// TIA Portal V15.1 export
// export: Created 2024-05-17T05:38:40.3336056Z, ExportSetting WithDefaults, DisplayName Totally Integrated Automation Portal, DisplayVersion V15.1 Update 5, DisplayName TIA Portal Openness, DisplayVersion V15.1 Update 5, DisplayName SINAMICS Startdrive Advanced, DisplayVersion V15.1, DisplayName G130, G150, S120, S150, SINAMICS MV, S210, DisplayVersion V15.1, DisplayName G110M, G120, G120C, G120D, G120P, DisplayVersion V15.1, DisplayName STEP 7 Professional, DisplayVersion V15.1 Update 5, DisplayName STEP 7 Safety, DisplayVersion V15.1, DisplayName WinCC Professional, DisplayVersion V15.1 Update 5, DisplayName SIMATIC Visualization Architect, DisplayVersion V15.1
FUNCTION "LGBHWPanelLedIndication" : Void   // FC6610, FBD
TITLE = LGBHWPanelLedIndication
{ S7_Optimized_Access := 'TRUE' }
VERSION : 0.1
// stored: AutoNumber false, IsIECCheckEnabled false, SetENOAutomatically False, UDAEnableTagReadback false
   VAR_INPUT
      I_NumberHMI : Int;   // Number of this HMI in the Modeselector
      I_ActiveHMI : Int;   // Active HMI in the Modeselector
      I_EStopAS_OK : Bool;   // Emergency Stop On AS Panel
      I_EStopZone_OK : Bool;   // Emergency Stop In The Safety Zone
      I_AlarmA : Bool;   // AlarmA
      I_AlarmB : Bool;   // AlarmB
      I_AlarmC : Bool;   // AlarmC
      I_Modes : "Modes";   // Modes
   END_VAR
   VAR_OUTPUT
      O_LED_Auto : Bool;   // Indication Automatic
      O_LED_Man : Bool;   // Indication Manual
      O_LED_Fault : Bool;   // Indication Fault
      O_LED_EStop : Bool;   // Indication Emergency Stop
   END_VAR
BEGIN

REGION Network 1: Indication Automatic
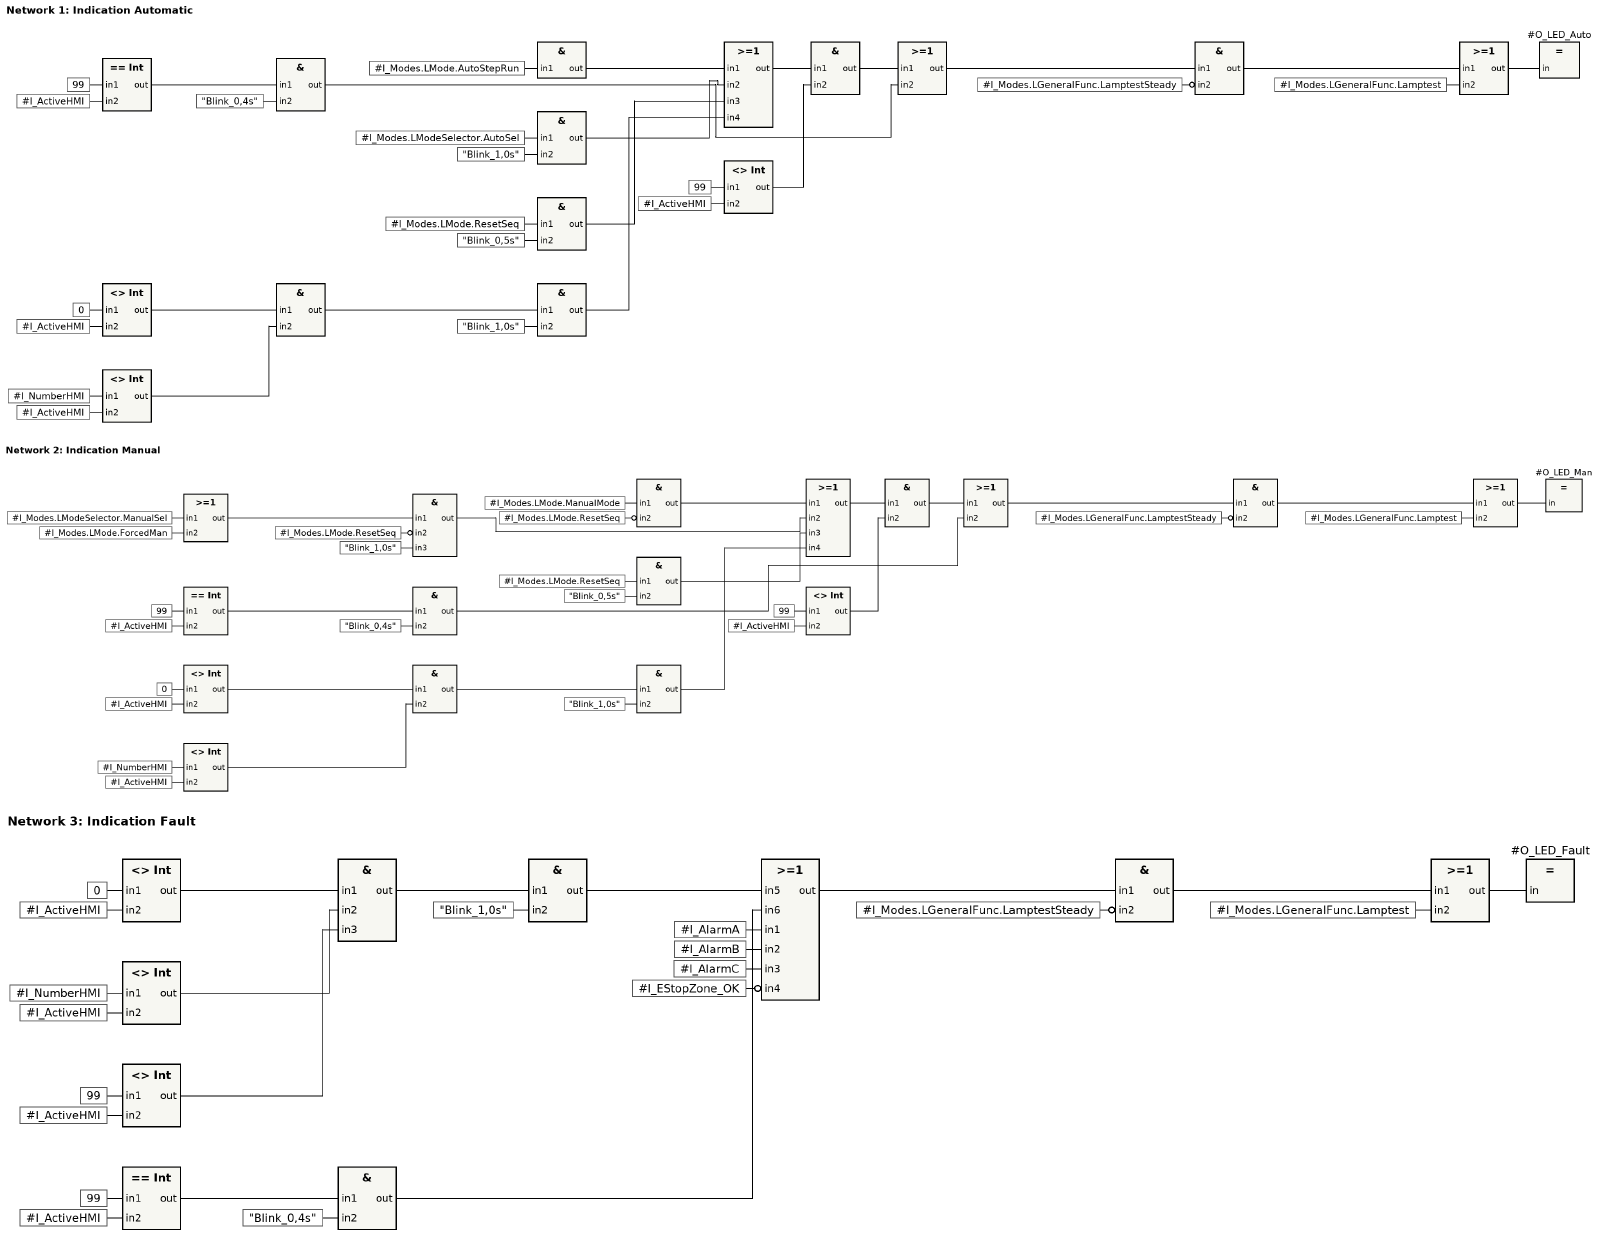
   #O_LED_Auto := ((((#I_Modes.LMode.AutoStepRun OR (#I_Modes.LModeSelector.AutoSel AND "Blink_1,0s") OR (#I_Modes.LMode.ResetSeq AND "Blink_0,5s") OR ((0 <> #I_ActiveHMI) AND (#I_NumberHMI <> #I_ActiveHMI) AND "Blink_1,0s")) AND (99 <> #I_ActiveHMI)) OR ((99 = #I_ActiveHMI) AND "Blink_0,4s")) AND NOT #I_Modes.LGeneralFunc.LamptestSteady) OR #I_Modes.LGeneralFunc.Lamptest;
END_REGION

REGION Network 2: Indication Manual
   #O_LED_Man := (((((#I_Modes.LMode.ManualMode AND NOT #I_Modes.LMode.ResetSeq) OR ((#I_Modes.LModeSelector.ManualSel OR #I_Modes.LMode.ForcedMan) AND NOT #I_Modes.LMode.ResetSeq AND "Blink_1,0s") OR (#I_Modes.LMode.ResetSeq AND "Blink_0,5s") OR ((0 <> #I_ActiveHMI) AND (#I_NumberHMI <> #I_ActiveHMI) AND "Blink_1,0s")) AND (99 <> #I_ActiveHMI)) OR ((99 = #I_ActiveHMI) AND "Blink_0,4s")) AND NOT #I_Modes.LGeneralFunc.LamptestSteady) OR #I_Modes.LGeneralFunc.Lamptest;
END_REGION

REGION Network 3: Indication Fault
   #O_LED_Fault := ((((0 <> #I_ActiveHMI) AND (#I_NumberHMI <> #I_ActiveHMI) AND (99 <> #I_ActiveHMI) AND "Blink_1,0s") OR ((99 = #I_ActiveHMI) AND "Blink_0,4s") OR #I_AlarmA OR #I_AlarmB OR #I_AlarmC OR NOT #I_EStopZone_OK) AND NOT #I_Modes.LGeneralFunc.LamptestSteady) OR #I_Modes.LGeneralFunc.Lamptest;
END_REGION

REGION Network 4: Indication Emergency Stop
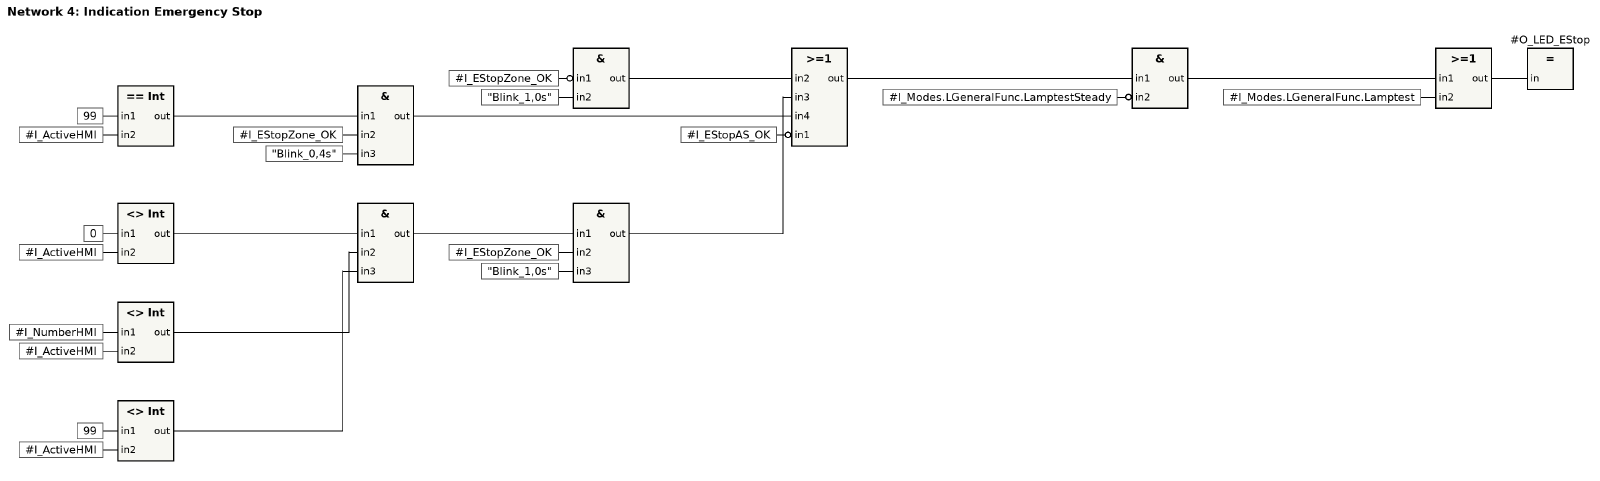
   #O_LED_EStop := (((NOT #I_EStopZone_OK AND "Blink_1,0s") OR ((0 <> #I_ActiveHMI) AND (#I_NumberHMI <> #I_ActiveHMI) AND (99 <> #I_ActiveHMI) AND #I_EStopZone_OK AND "Blink_1,0s") OR ((99 = #I_ActiveHMI) AND #I_EStopZone_OK AND "Blink_0,4s") OR NOT #I_EStopAS_OK) AND NOT #I_Modes.LGeneralFunc.LamptestSteady) OR #I_Modes.LGeneralFunc.Lamptest;
END_REGION
END_FUNCTION
